TYPE PRINTF_DATA : ARRAY [1..11]  OF STRING(LOG_SIZE);
END_TYPE

(* stored: Version 1.1.0.1, ProductVersion 3.1.4024.9
   DUT PRINTF_DATA: Id {c6d3bf89-572a-4f9f-a70b-19285d605cc9} *)
